TYPE T_NEST_OFFSET : ARRAY[1..MAX_MOVER]        OF
                     ARRAY[1..MAX_STATION_NEST] OF LREAL;
END_TYPE

(* stored: Version 1.1.0.1
   DUT T_NEST_OFFSET: Id {b6c19093-be05-4807-98f0-bb852377d37e} *)
